{attribute 'linkalways'} 
{attribute 'no_explicit_call' := 'This FB is a CLASS and must be accessed using methods or properties'}
{attribute 'enable_dynamic_creation'}
FUNCTION_BLOCK _ETcVnSvmSgdClassifierMarginType EXTENDS EnumDatatypeBase
VAR
	localData : ETcVnSvmSgdClassifierMarginType;
	activeData : REFERENCE TO ETcVnSvmSgdClassifierMarginType;
	enumBaseDatatype : _DINT(localData);
END_VAR

METHOD PRIVATE AddLocalEnumeration
VAR_INPUT
	Enumeration : T_MAXSTRING;
	Value : ETcVnSvmSgdClassifierMarginType;
END_VAR
AddEnumeration(Enumeration, Value);
END_METHOD

PROPERTY PUBLIC Address : PVOID
GET
Address := ADR(activeData);
END_GET
END_PROPERTY

METHOD PUBLIC ClearReference
VAR_INPUT
END_VAR
activeData REF= localData;
SetBaseDatatypeReference();
END_METHOD

METHOD PUBLIC Clone : I_Datatype
VAR
    pClone : POINTER TO _ETcVnSvmSgdClassifierMarginType;
END_VAR
pClone := __NEW(_ETcVnSvmSgdClassifierMarginType(InitialValue := Value));
Clone := pClone^;
END_METHOD

METHOD FB_init : BOOL
VAR_INPUT
	bInitRetains : BOOL; // if TRUE, the retain variables are initialized (warm start / cold start)
	bInCopyCode : BOOL;  // if TRUE, the instance afterwards gets moved into the copy code (online change)
	InitialValue : ETcVnSvmSgdClassifierMarginType;
END_VAR
localData := InitialValue;
AddBaseDatatype(enumBaseDatatype);
ClearReference();

AddLocalEnumeration('TCVN_SSCMT_SOFT_MARGIN', ETcVnSvmSgdClassifierMarginType.TCVN_SSCMT_SOFT_MARGIN);
AddLocalEnumeration('TCVN_SSCMT_HARD_MARGIN', ETcVnSvmSgdClassifierMarginType.TCVN_SSCMT_HARD_MARGIN);
END_METHOD

PROPERTY PUBLIC Identifier : T_MAXSTRING
GET
Identifier := 'ETcVnSvmSgdClassifierMarginType';
END_GET
END_PROPERTY

METHOD IsEnumeratorValueEqual : BOOL
VAR_INPUT
	Enumerator : I_KeyValueForwardEnumerator;
END_VAR
VAR
	storedValue : ETcVnSvmSgdClassifierMarginType;
END_VAR
IF NOT Enumerator.TryGet(storedValue) THEN
	RETURN;
END_IF

IsEnumeratorValueEqual := storedValue = activeData;
END_METHOD

METHOD PUBLIC MakeReferenceTo
VAR_INPUT
	ReferenceTarget : REFERENCE TO ETcVnSvmSgdClassifierMarginType;
END_VAR
activeData REF= ReferenceTarget;
SetBaseDatatypeReference();
END_METHOD

METHOD PROTECTED SetBaseDatatypeReference
VAR_INPUT
END_VAR
enumBaseDatatype.MakeReferenceTo(activeData);
END_METHOD

PROPERTY PUBLIC Size : UDINT
GET
Size := SIZEOF(activeData);
END_GET
END_PROPERTY

METHOD TryMakeReferenceTo : BOOL
VAR_INPUT
	Target : I_Datatype;
END_VAR
VAR
	targetAsEnum : I_EnumDatatype;
	pTargetData : POINTER TO ETcVnSvmSgdClassifierMarginType;
END_VAR
IF NOT Target.TryResolveAsEnumDatatype(targetAsEnum) THEN
	RETURN;
END_IF

IF targetAsEnum.Identifier <> Identifier THEN
	RETURN;
END_IF

pTargetData := Target.Address;
activeData REF= pTargetData^;
SetBaseDatatypeReference();
TryMakeReferenceTo := TRUE;
END_METHOD

PROPERTY PUBLIC Value : ETcVnSvmSgdClassifierMarginType
GET
Value := activeData;
END_GET
SET
activeData := Value;
END_SET
END_PROPERTY

END_FUNCTION_BLOCK

(* stored: Version 1.1.0.1
   POU _ETcVnSvmSgdClassifierMarginType: Id {f088a38f-7276-4946-b6f5-dd4e81c97920}, SpecialFunc None
   Folder Constructor: Id {f1cb38d2-c646-450d-964f-0e2751dafee7}
   Folder Private: Id {c7bad6c3-ca83-4ce9-adea-7b911fc7272e}
   Folder Protected: Id {a15265f9-7543-49c7-b4cb-2ee27fa73db7}
   Method AddLocalEnumeration: Id {12340b7e-48ba-4982-9cc7-f968e6324839}
   Property Address: Id {72732472-6dba-45d0-a13f-808932fa457d}
   Get Get: Id {e06b9d5d-3d8f-4209-a1bf-ce56adf091d2}
   Method ClearReference: Id {22a8d02e-eb72-405c-9aeb-0517c0a7cf3c}
   Method Clone: Id {e8f5f81c-2b38-493d-90fc-9fcd7c28b75e}
   Method FB_init: Id {66cbd0cd-82c4-4f1d-a8f0-014c05c64e41}
   Property Identifier: Id {c485ffa8-9546-40f7-a5bc-fd28c6e994a0}
   Get Get: Id {9610138f-eae5-4516-b78a-52460b3455af}
   Method IsEnumeratorValueEqual: Id {d8d58746-3d4d-45d6-b681-5a094425e506}
   Method MakeReferenceTo: Id {30e81590-6444-43ab-a2b9-cd96a290fc8d}
   Method SetBaseDatatypeReference: Id {c5c01bbb-399f-4f8a-bd91-d501d785a36f}
   Property Size: Id {a49d0442-f590-4463-b35f-fe9db6077cce}
   Get Get: Id {92422514-97af-409a-8cb7-1ce6abd5ff3c}
   Method TryMakeReferenceTo: Id {6ac11203-0634-475b-8a03-451c63244a7d}
   Property Value: Id {dfbf3154-b2de-4c72-a81e-a3858208e55a}
   Get Get: Id {c8499673-d0af-4fa5-b18a-222919446a5c}
   Set Set: Id {a85a84d1-964c-4ff7-8864-5691832f0345} *)
